Omron CX-Programmer project NewProject (CX-Programmer 9.75)

# PLC NewPLC1: CP1E N40

## Global symbols (name address type ; comment)
0.00 BOOL  ; REED7.1
0.01 BOOL  ; REED7.2
0.02 BOOL  ; REED8.1
0.03 BOOL  ; REED8.2
0.04 BOOL  ; REED9.1
0.05 BOOL  ; REED9.2
0.06 BOOL  ; REED8.3
0.07 BOOL  ; REED7.3
0.08 BOOL  ; REED11.1
0.09 BOOL  ; REED11.2
0.10 BOOL  ; REED12.1
0.11 BOOL  ; REED12.2
100.01 BOOL  ; ACT2-OUT
100.02 BOOL  ; ACT3-OUT
100.03 BOOL  ; ACT4-OUT
100.04 BOOL  ; ACT5-OUT
100.05 BOOL  ; ACT6-OUT
100.06 BOOL  ; ACT1-OUT
100.07 BOOL  ; ACT7-OUT
101.00 BOOL  ; ACT8-OUT
101.01 BOOL  ; ACT9-OUT
101.02 BOOL  ; ACT10-OUT
101.03 BOOL  ; ACT11-OUT
101.04 BOOL  ; ACT12-OUT
101.07 BOOL  ; SAFTY VALVE
1.01 BOOL  ; REED10.1
1.02 BOOL  ; REED10.2
1.03 BOOL  ; REED 1.1
1.04 BOOL  ; REED 1.2
1.05 BOOL  ; REED 2.1
1.06 BOOL  ; REED 2.2
1.07 BOOL  ; REED 3.1
1.08 BOOL  ; REED 3.2
1.09 BOOL  ; REED 6.1
1.10 BOOL  ; REED 6.2
1.11 BOOL  ; EM STOP
2.01 BOOL  ; RUN
T000 BOOL  ; TIMER1
T001 BOOL  ; TIMER2
T003 BOOL  ; MANUAL TIMER
T004 BOOL  ; ACT4-TIMER
W0.00 BOOL  ; START_HMI
W0.01 BOOL  ; STOP_HMI
W0.02 BOOL  ; RUN
W1.11 BOOL  ; EM_STOP_HMI
W2.00 BOOL  ; POWER
W30.00 BOOL  ; ACT2
W30.01 BOOL  ; ACT3
W30.02 BOOL  ; ACT4
W30.03 BOOL  ; ACT1
W30.04 BOOL  ; ACT7
W30.05 BOOL  ; ACT8
W30.06 BOOL  ; ACT9
W30.07 BOOL  ; ACT10
W30.08 BOOL  ; ACT11
W30.09 BOOL  ; ACT12
W31.00 BOOL  ; ACT5
W31.01 BOOL  ; ACT6
W35.00 BOOL  ; FRONT-SET
W35.01 BOOL  ; BACK-SET
W36.00 BOOL  ; INITIAL_DONE
W44.00 BOOL  ; BED_LATCH
W44.01 BOOL  ; RUN_LATCH
W45.00 BOOL  ; LATCH_10
W45.01 BOOL  ; DOWN_LATCH
W4.00 BOOL  ; ACT4-SET
W4.01 BOOL  ; ACT4-RESET
W5.01 BOOL  ; FRONT
W5.02 BOOL  ; BACK
W5.03 BOOL  ; STEP
W5.05 BOOL  ; STEP01
W70.00 BOOL  ; R7.1
W70.01 BOOL  ; R7.2
W70.02 BOOL  ; R8.1
W70.03 BOOL  ; R8.2
W70.04 BOOL  ; R9.1
W70.05 BOOL  ; R9.2
W70.06 BOOL  ; R8.3
W70.07 BOOL  ; R7.3
W70.08 BOOL  ; R11.1
W70.09 BOOL  ; R11.2
W71.00 BOOL  ; R12.1
W71.01 BOOL  ; R12.2
W71.02 BOOL  ; R10.1
W71.03 BOOL  ; R10.2
W71.04 BOOL  ; R1.1
W71.05 BOOL  ; R1.2
W71.06 BOOL  ; R2.1
W71.07 BOOL  ; R2.2
W71.08 BOOL  ; R3.1
W71.09 BOOL  ; R3.2
W72.00 BOOL  ; R6.1
W72.01 BOOL  ; R6.2

## Program NewProgram1 (cyclic task 0)

### Section MAIN01

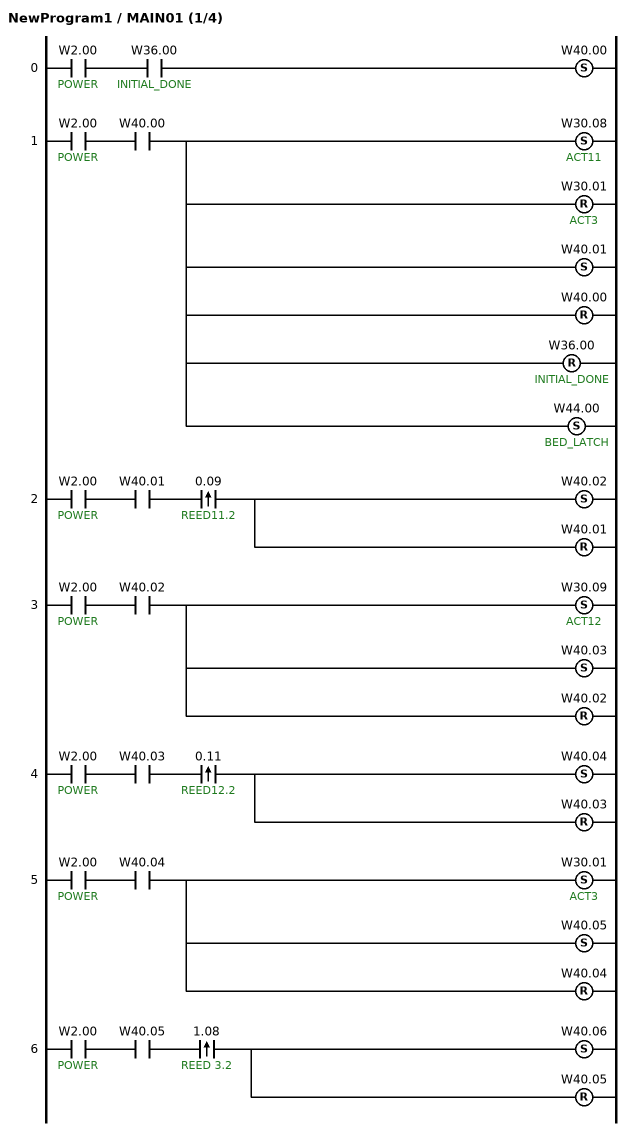
; rung 0
LD W2.00  ; POWER
AND W36.00  ; INITIAL_DONE
SET W40.00
; rung 1
LD W2.00  ; POWER
AND W40.00
SET W30.08  ; ACT11
RSET W30.01  ; ACT3
SET W40.01
RSET W40.00
RSET W36.00  ; INITIAL_DONE
SET W44.00  ; BED_LATCH
; rung 2
LD W2.00  ; POWER
AND W40.01
@AND 0.09  ; REED11.2
SET W40.02
RSET W40.01
; rung 3
LD W2.00  ; POWER
AND W40.02
SET W30.09  ; ACT12
SET W40.03
RSET W40.02
; rung 4
LD W2.00  ; POWER
AND W40.03
@AND 0.11  ; REED12.2
SET W40.04
RSET W40.03
; rung 5
LD W2.00  ; POWER
AND W40.04
SET W30.01  ; ACT3
SET W40.05
RSET W40.04
; rung 6
LD W2.00  ; POWER
AND W40.05
@AND 1.08  ; REED 3.2
SET W40.06
RSET W40.05

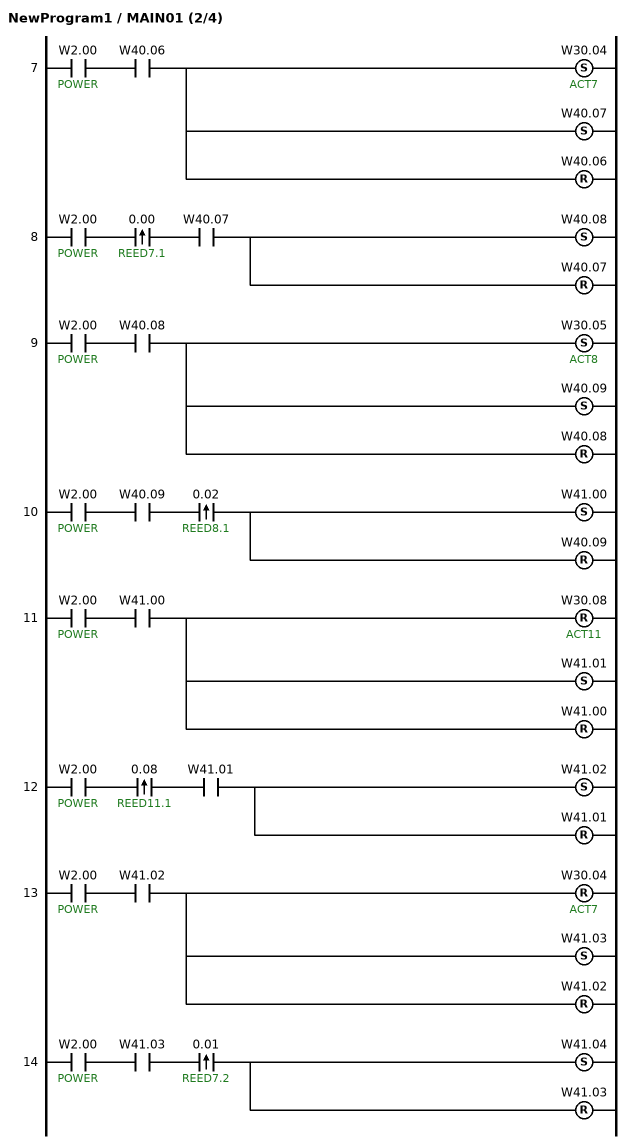
; rung 7
LD W2.00  ; POWER
AND W40.06
SET W30.04  ; ACT7
SET W40.07
RSET W40.06
; rung 8
LD W2.00  ; POWER
@AND 0.00  ; REED7.1
AND W40.07
SET W40.08
RSET W40.07
; rung 9
LD W2.00  ; POWER
AND W40.08
SET W30.05  ; ACT8
SET W40.09
RSET W40.08
; rung 10
LD W2.00  ; POWER
AND W40.09
@AND 0.02  ; REED8.1
SET W41.00
RSET W40.09
; rung 11
LD W2.00  ; POWER
AND W41.00
RSET W30.08  ; ACT11
SET W41.01
RSET W41.00
; rung 12
LD W2.00  ; POWER
@AND 0.08  ; REED11.1
AND W41.01
SET W41.02
RSET W41.01
; rung 13
LD W2.00  ; POWER
AND W41.02
RSET W30.04  ; ACT7
SET W41.03
RSET W41.02
; rung 14
LD W2.00  ; POWER
AND W41.03
@AND 0.01  ; REED7.2
SET W41.04
RSET W41.03

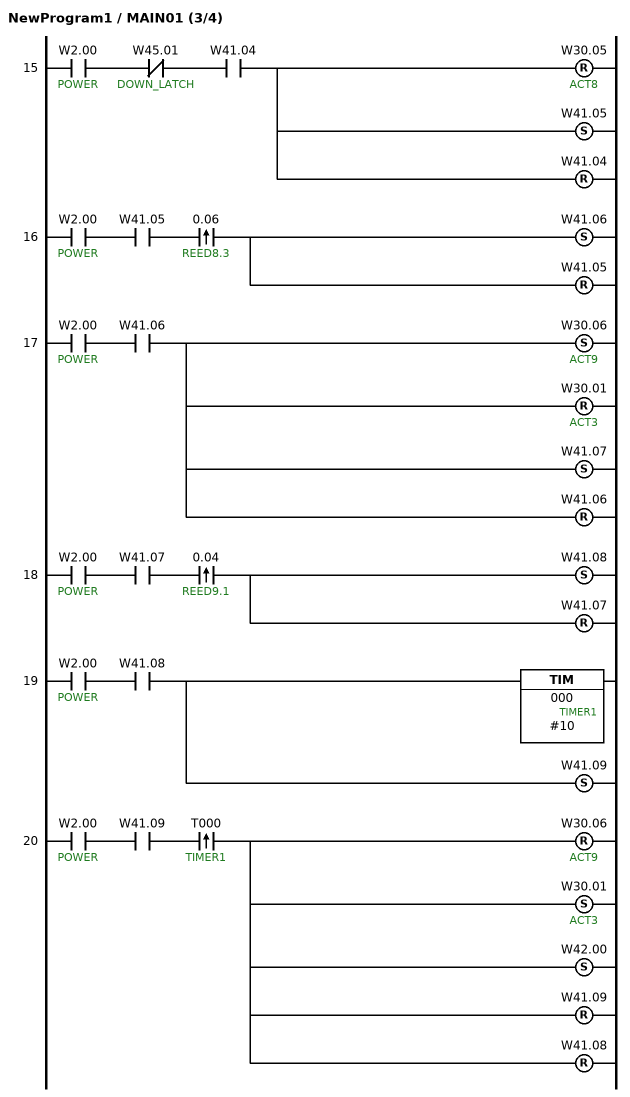
; rung 15
LD W2.00  ; POWER
ANDNOT W45.01  ; DOWN_LATCH
AND W41.04
RSET W30.05  ; ACT8
SET W41.05
RSET W41.04
; rung 16
LD W2.00  ; POWER
AND W41.05
@AND 0.06  ; REED8.3
SET W41.06
RSET W41.05
; rung 17
LD W2.00  ; POWER
AND W41.06
SET W30.06  ; ACT9
RSET W30.01  ; ACT3
SET W41.07
RSET W41.06
; rung 18
LD W2.00  ; POWER
AND W41.07
@AND 0.04  ; REED9.1
SET W41.08
RSET W41.07
; rung 19
LD W2.00  ; POWER
AND W41.08
TIM 000 #10  ; TIMER1
SET W41.09
; rung 20
LD W2.00  ; POWER
AND W41.09
@AND T000  ; TIMER1
RSET W30.06  ; ACT9
SET W30.01  ; ACT3
SET W42.00
RSET W41.09
RSET W41.08

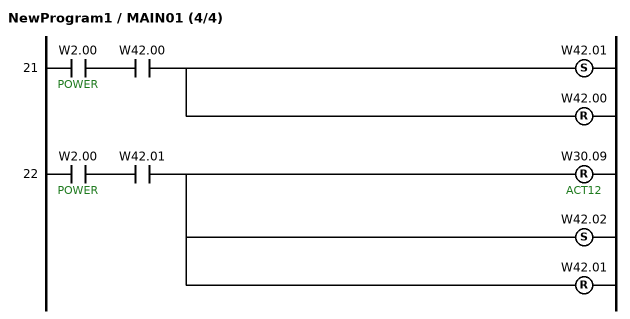
; rung 21
LD W2.00  ; POWER
AND W42.00
SET W42.01
RSET W42.00
; rung 22
LD W2.00  ; POWER
AND W42.01
RSET W30.09  ; ACT12
SET W42.02
RSET W42.01

### Section MAIN02

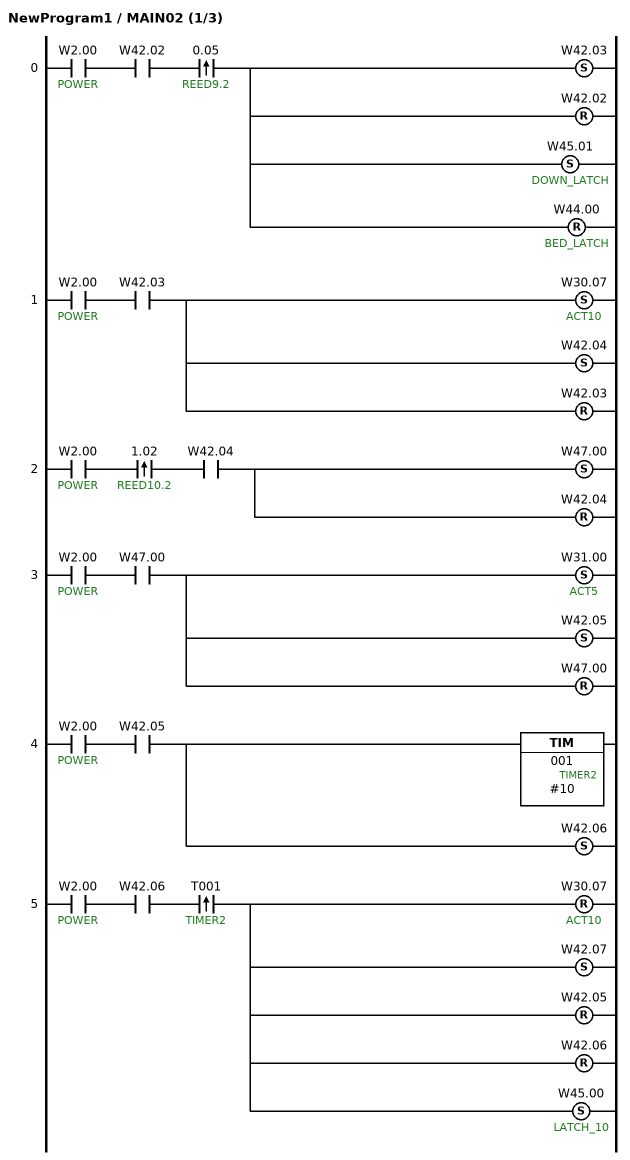
; rung 0
LD W2.00  ; POWER
AND W42.02
@AND 0.05  ; REED9.2
SET W42.03
RSET W42.02
SET W45.01  ; DOWN_LATCH
RSET W44.00  ; BED_LATCH
; rung 1
LD W2.00  ; POWER
AND W42.03
SET W30.07  ; ACT10
SET W42.04
RSET W42.03
; rung 2
LD W2.00  ; POWER
@AND 1.02  ; REED10.2
AND W42.04
SET W47.00
RSET W42.04
; rung 3
LD W2.00  ; POWER
AND W47.00
SET W31.00  ; ACT5
SET W42.05
RSET W47.00
; rung 4
LD W2.00  ; POWER
AND W42.05
TIM 001 #10  ; TIMER2
SET W42.06
; rung 5
LD W2.00  ; POWER
AND W42.06
@AND T001  ; TIMER2
RSET W30.07  ; ACT10
SET W42.07
RSET W42.05
RSET W42.06
SET W45.00  ; LATCH_10

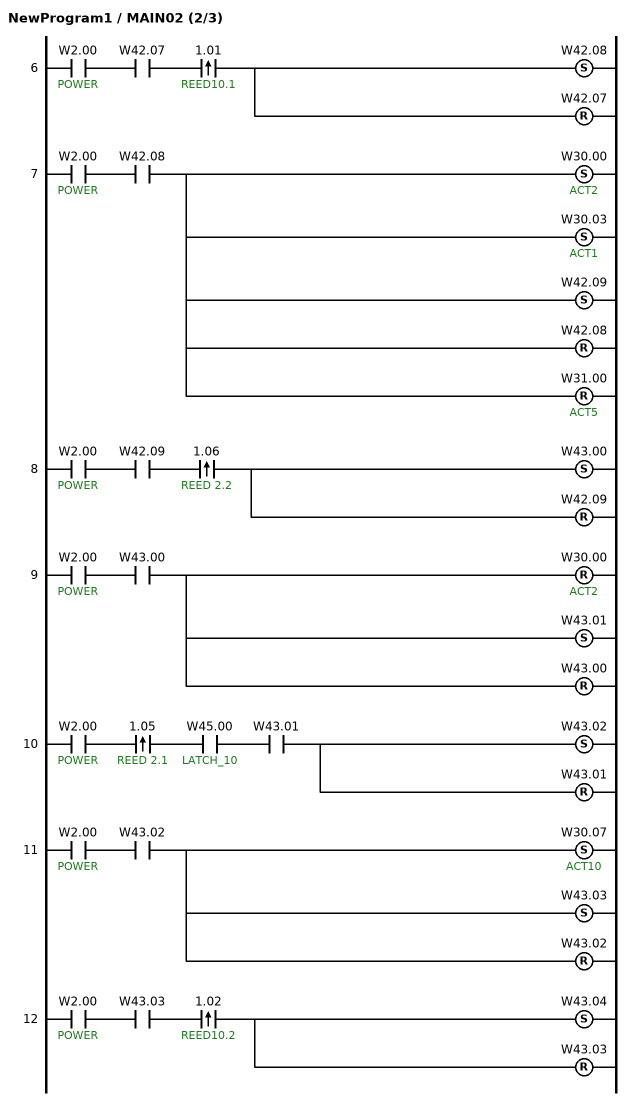
; rung 6
LD W2.00  ; POWER
AND W42.07
@AND 1.01  ; REED10.1
SET W42.08
RSET W42.07
; rung 7
LD W2.00  ; POWER
AND W42.08
SET W30.00  ; ACT2
SET W30.03  ; ACT1
SET W42.09
RSET W42.08
RSET W31.00  ; ACT5
; rung 8
LD W2.00  ; POWER
AND W42.09
@AND 1.06  ; REED 2.2
SET W43.00
RSET W42.09
; rung 9
LD W2.00  ; POWER
AND W43.00
RSET W30.00  ; ACT2
SET W43.01
RSET W43.00
; rung 10
LD W2.00  ; POWER
@AND 1.05  ; REED 2.1
AND W45.00  ; LATCH_10
AND W43.01
SET W43.02
RSET W43.01
; rung 11
LD W2.00  ; POWER
AND W43.02
SET W30.07  ; ACT10
SET W43.03
RSET W43.02
; rung 12
LD W2.00  ; POWER
AND W43.03
@AND 1.02  ; REED10.2
SET W43.04
RSET W43.03

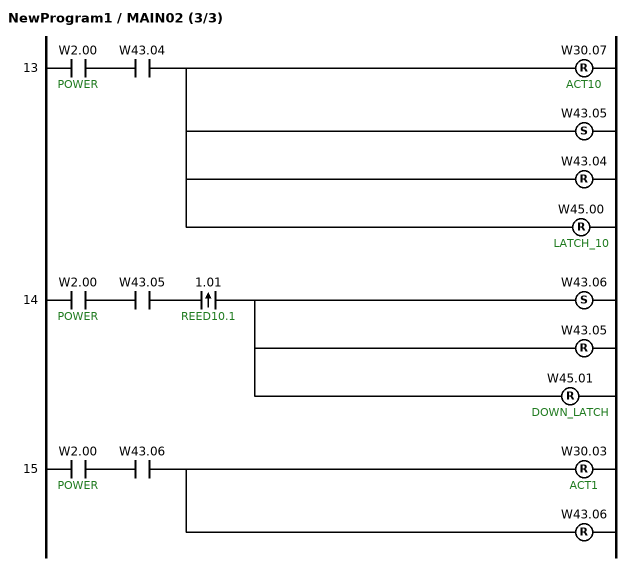
; rung 13
LD W2.00  ; POWER
AND W43.04
RSET W30.07  ; ACT10
SET W43.05
RSET W43.04
RSET W45.00  ; LATCH_10
; rung 14
LD W2.00  ; POWER
AND W43.05
@AND 1.01  ; REED10.1
SET W43.06
RSET W43.05
RSET W45.01  ; DOWN_LATCH
; rung 15
LD W2.00  ; POWER
AND W43.06
RSET W30.03  ; ACT1
RSET W43.06

### Section INITIAL

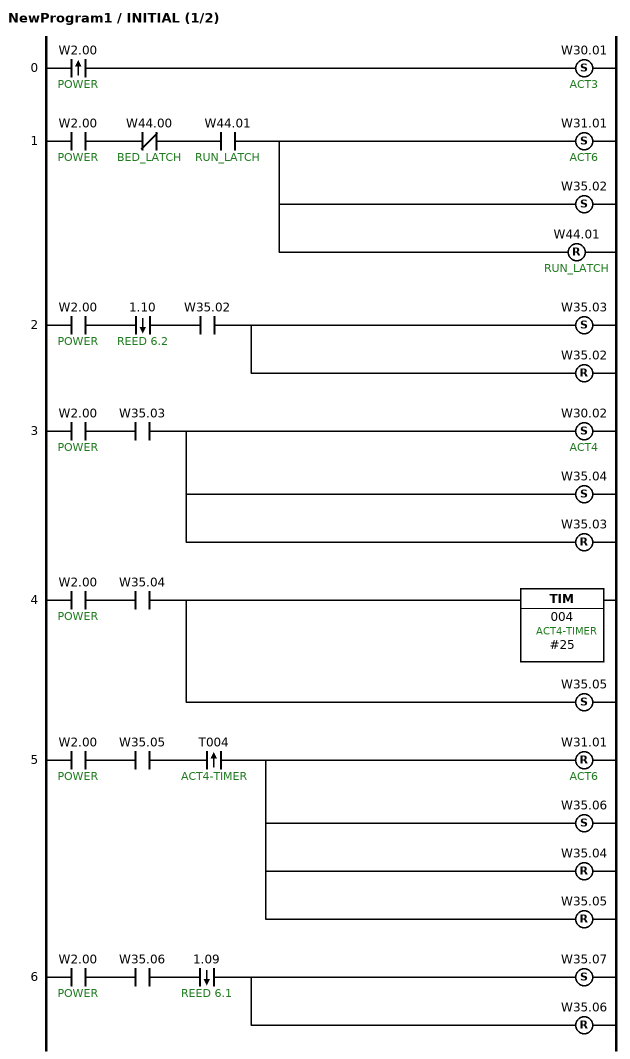
; rung 0
@LD W2.00  ; POWER
SET W30.01  ; ACT3
; rung 1
LD W2.00  ; POWER
ANDNOT W44.00  ; BED_LATCH
AND W44.01  ; RUN_LATCH
SET W31.01  ; ACT6
SET W35.02
RSET W44.01  ; RUN_LATCH
; rung 2
LD W2.00  ; POWER
%AND 1.10  ; REED 6.2
AND W35.02
SET W35.03
RSET W35.02
; rung 3
LD W2.00  ; POWER
AND W35.03
SET W30.02  ; ACT4
SET W35.04
RSET W35.03
; rung 4
LD W2.00  ; POWER
AND W35.04
TIM 004 #25  ; ACT4-TIMER
SET W35.05
; rung 5
LD W2.00  ; POWER
AND W35.05
@AND T004  ; ACT4-TIMER
RSET W31.01  ; ACT6
SET W35.06
RSET W35.04
RSET W35.05
; rung 6
LD W2.00  ; POWER
AND W35.06
%AND 1.09  ; REED 6.1
SET W35.07
RSET W35.06

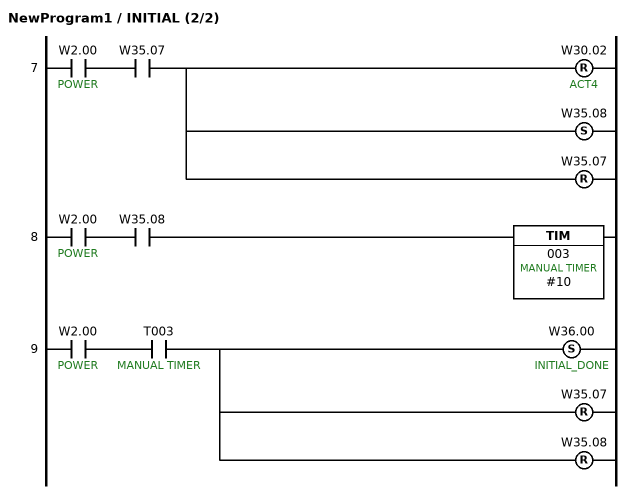
; rung 7
LD W2.00  ; POWER
AND W35.07
RSET W30.02  ; ACT4
SET W35.08
RSET W35.07
; rung 8
LD W2.00  ; POWER
AND W35.08
TIM 003 #10  ; MANUAL TIMER
; rung 9
LD W2.00  ; POWER
AND T003  ; MANUAL TIMER
SET W36.00  ; INITIAL_DONE
RSET W35.07
RSET W35.08

### Section POWER

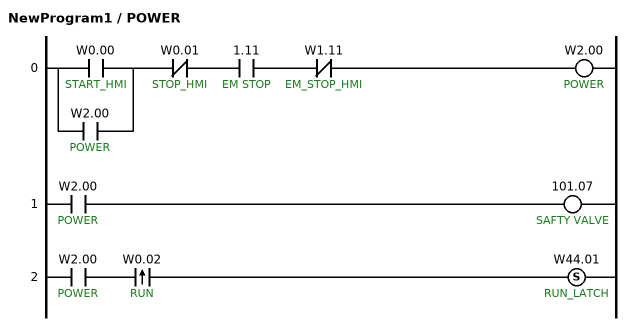
; rung 0
LD W0.00  ; START_HMI
OR W2.00  ; POWER
ANDNOT W0.01  ; STOP_HMI
AND 1.11  ; EM STOP
ANDNOT W1.11  ; EM_STOP_HMI
OUT W2.00  ; POWER
; rung 1
LD W2.00  ; POWER
OUT 101.07  ; SAFTY VALVE
; rung 2
LD W2.00  ; POWER
@AND W0.02  ; RUN
SET W44.01  ; RUN_LATCH

### Section OUTPUT

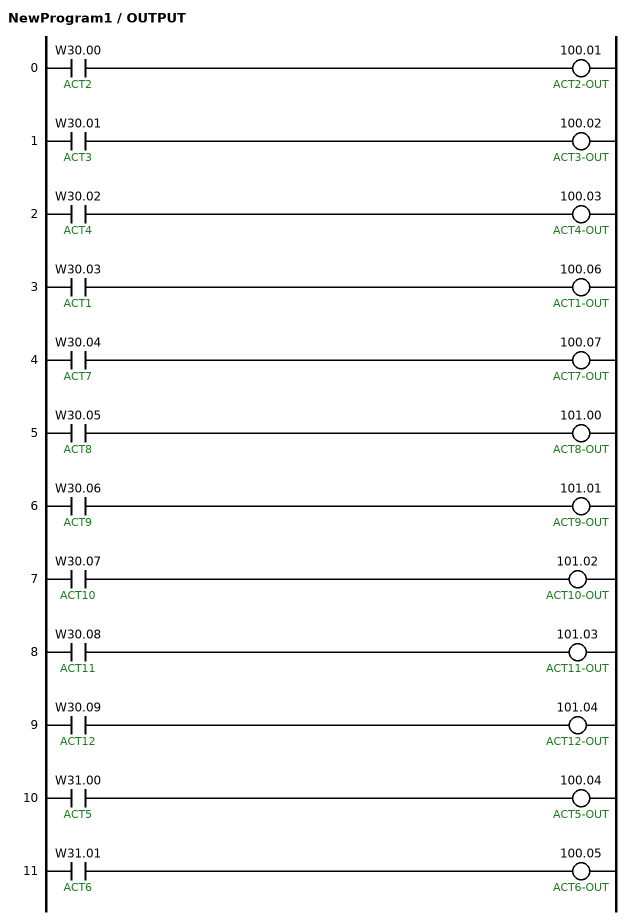
; rung 0
LD W30.00  ; ACT2
OUT 100.01  ; ACT2-OUT
; rung 1
LD W30.01  ; ACT3
OUT 100.02  ; ACT3-OUT
; rung 2
LD W30.02  ; ACT4
OUT 100.03  ; ACT4-OUT
; rung 3
LD W30.03  ; ACT1
OUT 100.06  ; ACT1-OUT
; rung 4
LD W30.04  ; ACT7
OUT 100.07  ; ACT7-OUT
; rung 5
LD W30.05  ; ACT8
OUT 101.00  ; ACT8-OUT
; rung 6
LD W30.06  ; ACT9
OUT 101.01  ; ACT9-OUT
; rung 7
LD W30.07  ; ACT10
OUT 101.02  ; ACT10-OUT
; rung 8
LD W30.08  ; ACT11
OUT 101.03  ; ACT11-OUT
; rung 9
LD W30.09  ; ACT12
OUT 101.04  ; ACT12-OUT
; rung 10
LD W31.00  ; ACT5
OUT 100.04  ; ACT5-OUT
; rung 11
LD W31.01  ; ACT6
OUT 100.05  ; ACT6-OUT

### Section INPUT

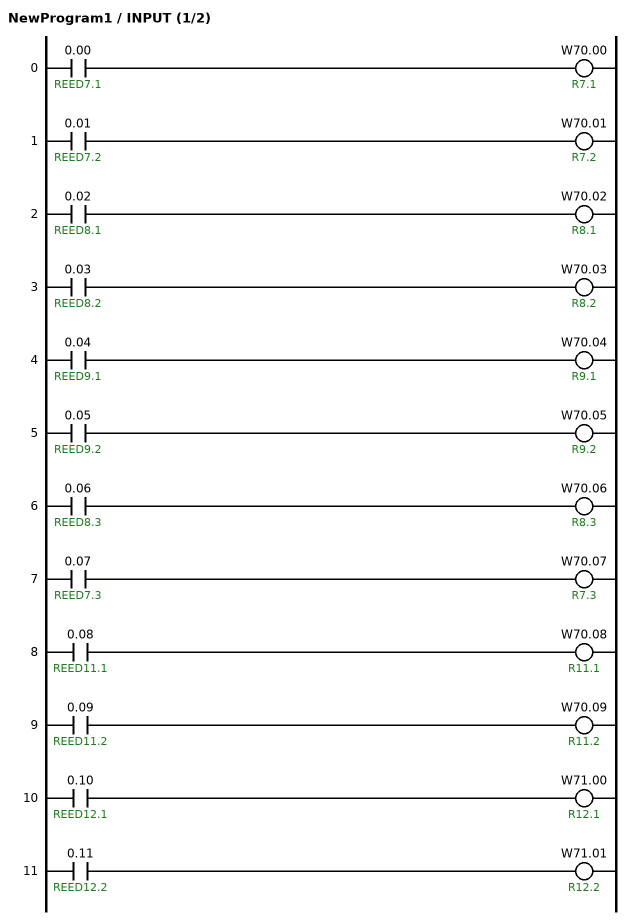
; rung 0
LD 0.00  ; REED7.1
OUT W70.00  ; R7.1
; rung 1
LD 0.01  ; REED7.2
OUT W70.01  ; R7.2
; rung 2
LD 0.02  ; REED8.1
OUT W70.02  ; R8.1
; rung 3
LD 0.03  ; REED8.2
OUT W70.03  ; R8.2
; rung 4
LD 0.04  ; REED9.1
OUT W70.04  ; R9.1
; rung 5
LD 0.05  ; REED9.2
OUT W70.05  ; R9.2
; rung 6
LD 0.06  ; REED8.3
OUT W70.06  ; R8.3
; rung 7
LD 0.07  ; REED7.3
OUT W70.07  ; R7.3
; rung 8
LD 0.08  ; REED11.1
OUT W70.08  ; R11.1
; rung 9
LD 0.09  ; REED11.2
OUT W70.09  ; R11.2
; rung 10
LD 0.10  ; REED12.1
OUT W71.00  ; R12.1
; rung 11
LD 0.11  ; REED12.2
OUT W71.01  ; R12.2

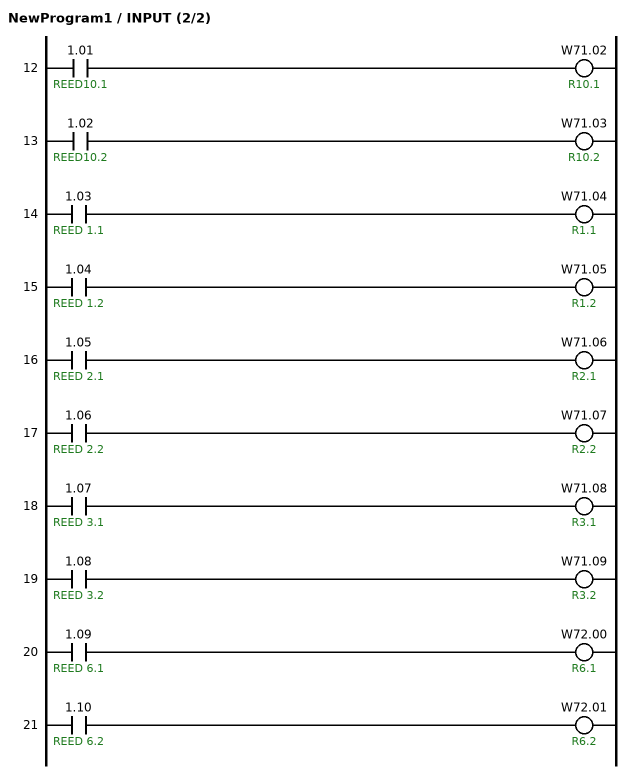
; rung 12
LD 1.01  ; REED10.1
OUT W71.02  ; R10.1
; rung 13
LD 1.02  ; REED10.2
OUT W71.03  ; R10.2
; rung 14
LD 1.03  ; REED 1.1
OUT W71.04  ; R1.1
; rung 15
LD 1.04  ; REED 1.2
OUT W71.05  ; R1.2
; rung 16
LD 1.05  ; REED 2.1
OUT W71.06  ; R2.1
; rung 17
LD 1.06  ; REED 2.2
OUT W71.07  ; R2.2
; rung 18
LD 1.07  ; REED 3.1
OUT W71.08  ; R3.1
; rung 19
LD 1.08  ; REED 3.2
OUT W71.09  ; R3.2
; rung 20
LD 1.09  ; REED 6.1
OUT W72.00  ; R6.1
; rung 21
LD 1.10  ; REED 6.2
OUT W72.01  ; R6.2

### Section END
; rung 0
END(001)